Fanuc KAREL source: KT00962.KL

PROGRAM KT00962
%NOLOCKGROUP
VAR
  ENTRY: INTEGER
  PNAME: STRING[80]
  VNAME: STRING[80]
  STATUS: INTEGER
  VALUE: POSITION
BEGIN
  ENTRY = 0
  PNAME = ''
  VNAME = 'VALUE'
  SET_VAR(ENTRY, PNAME, VNAME, VALUE, STATUS)
END KT00962
